// TIA Portal project "学习利用循环指令跑马灯_V16" (V16)

(* hardware
DEVICE "S7-1200 station_1"  S7-1200 Station
   slot 0: "Rack_0"  S7-1200 Rack  Rack  V1.0
   slot 1: "PLC_1"  CPU 1214C DC/DC/DC  6ES7 214-1AG40-0XB0  V4.2
*)

// ===== PLC "PLC_1"  CPU 1214C DC/DC/DC =====

VAR_GLOBAL   // PLC tag table "默认变量表"
   "Tag_1" AT %M0.0 : Bool;
   "Tag_2" AT %M0.1 : Bool;
   "Tag_3" AT %M0.3 : Bool;
   "Tag_4" AT %MD100 : Time;
   "Tag_5" AT %M0.4 : Bool;
   "Tag_6" AT %M0.5 : Bool;
   "Tag_7" AT %QB10 : Byte;
   "Tag_8" AT %M0.7 : Bool;
END_VAR

// folder: System blocks/Program resources

DATA_BLOCK "IEC_Timer_0_DB"   // DB1
{ S7_Optimized_Access := 'TRUE' }
AUTHOR : Simatic
FAMILY : IEC
NAME : IEC_TMR
VERSION : 1.0
// stored: InstanceOfName IEC_TIMER
"IEC_TIMER"
BEGIN
END_DATA_BLOCK

// folder: (top level)

ORGANIZATION_BLOCK "Main"   // OB1, LAD, ProgramCycle
TITLE = "Main Program Sweep (Cycle)"
{ S7_Optimized_Access := 'TRUE' }
VERSION : 0.1
   VAR_INPUT
      Initial_Call : Bool;   // Initial call of this OB
      Remanence : Bool;   // =True, if remanent data are available
   END_VAR
   VAR_TEMP   // added for the SCL form of the ladder/FBD networks
      _w1 : Bool;
   END_VAR
BEGIN

REGION Network 1
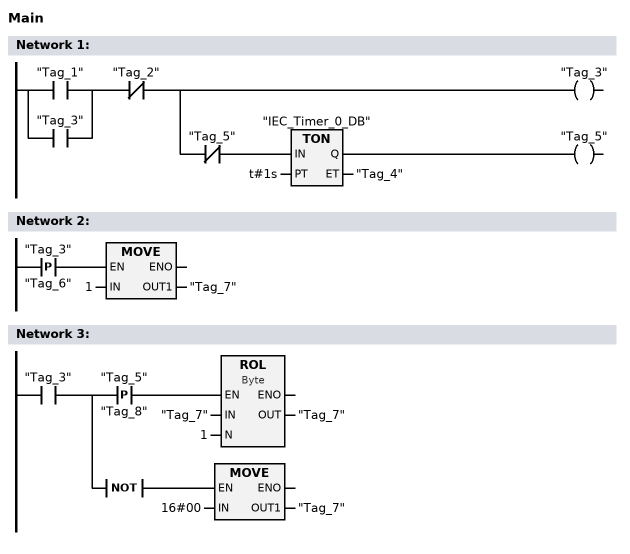
   "Tag_3" := ("Tag_1" OR "Tag_3") AND NOT "Tag_2";
   "IEC_Timer_0_DB".TON(IN := "Tag_3" AND NOT "Tag_5", PT := t#1s, ET => "Tag_4");
   "Tag_5" := "IEC_Timer_0_DB".Q;
END_REGION

REGION Network 2
   RUNG wire#powerrail
      P_Contact(operand := "Tag_3", bit := "Tag_6")
      Move(in := 1, out1 => "Tag_7")
   END_RUNG
   // the same network as SCL:
   #_w1 := "Tag_3" AND NOT "Tag_6";   // rising edge of "Tag_3"
   "Tag_6" := "Tag_3";
   IF #_w1 THEN "Tag_7" := 1; END_IF;
END_REGION

REGION Network 3
   #_w1 := "Tag_3" AND "Tag_5" AND NOT "Tag_8";   // rising edge of "Tag_5"
   "Tag_8" := "Tag_5";
   IF #_w1 THEN "Tag_7" := ROL(IN := "Tag_7", N := 1); END_IF;
   IF NOT "Tag_3" THEN "Tag_7" := 16#00; END_IF;
END_REGION
END_ORGANIZATION_BLOCK